PROGRAM MAIN
VAR
	value: uint;
END_VAR

END_PROGRAM

(* stored: Version 1.1.0.1, ProductVersion 3.1.4024.4
   POU MAIN: Id {e217a535-3330-4e80-92d4-a155d5b6d80b}, SpecialFunc None *)
